FUNCTION_BLOCK FB_Actuator_NoFeedback
VAR
	AdvanceOUT		: FB_DigitalOutput;
	RetractOUT		: FB_DigitalOutput;
	
	AdvanceBit			: BOOL := FALSE;
	RetractBit			: BOOL := FALSE;
	
	Advanced		: BOOL := FALSE;
	Retracted		: BOOL := FALSE;
	
	AdvanceTimer	: TON;
	RetractTimer	: TON;
END_VAR

AdvanceOUT();
RetractOUT();

AdvanceTimer(IN := AdvanceBit, PT := T#0.06S);
AdvanceOUT.SetOutput(AdvanceTimer.Q);
Advanced := AdvanceOUT.P_Output;

RetractTimer(IN := RetractBit, PT := T#0.06S);
RetractOUT.SetOutput(RetractTimer.Q);
Retracted := RetractOUT.P_Output;

METHOD PUBLIC Advance : BOOL
RetractOUT.SetOutput(FALSE);
RetractBit := FALSE;
Advance := TRUE;
END_METHOD

PROPERTY P_Advanced : BOOL
GET
P_Advanced := Advanced;
END_GET
END_PROPERTY

PROPERTY P_Retracted : BOOL
GET
P_Retracted := Retracted;
END_GET
END_PROPERTY

METHOD PUBLIC Retract : BOOL
AdvanceOUT.SetOutput(FALSE);
Retract := TRUE;
AdvanceBit := FALSE;
END_METHOD

END_FUNCTION_BLOCK

(* stored: Version 1.1.0.1
   POU FB_Actuator_NoFeedback: Id {961f5635-0748-4d42-a48e-76bb5fb40e45}, SpecialFunc None
   Folder Methods: Id {bdd8ad22-4375-4ffc-b229-f074dd9c4af4}
   Folder Properties: Id {ab013551-f43d-4387-b701-c63914ec184a}
   Method Advance: Id {a130657e-8b41-4df2-b160-32a3e49d213c}
   Property P_Advanced: Id {af95aa15-9288-40d6-8172-f305b3908d89}
   Get Get: Id {c970a032-32a7-4450-89f4-27cb6eef00c2}
   Property P_Retracted: Id {310df0ce-3fcd-4a40-9448-568383b77778}
   Get Get: Id {97a67513-e1f0-4d7b-b95e-ee5375389c57}
   Method Retract: Id {dd9f7d52-b76a-457a-abbe-88f9c9c8ffcb} *)
